// TIA Portal V16 export
// export: Created 2024-12-03T15:41:41.5093467Z, ExportSetting WithDefaults, DisplayName Totally Integrated Automation Portal, DisplayVersion V16 Update 6, DisplayName TIA Portal Version Control Interface, DisplayVersion V16 Update 2, DisplayName TIA Portal Openness, DisplayVersion V16 Update 6, DisplayName TIA Portal Teamcenter Gateway, DisplayVersion V16, DisplayName SINAMICS Startdrive Advanced, DisplayVersion V16 Update 5, DisplayName SINAMICS Startdrive G130, G150, S120, S150, SINAMICS MV, S210, DisplayVersion V16 Update 5, DisplayName SINAMICS Startdrive G110M, G120, G120C, G120D, G120P, G115D, DisplayVersion V16 Update 5, DisplayName STEP 7 Professional, DisplayVersion V16 Update 6, DisplayName STEP 7 Safety, DisplayVersion V16, DisplayName WinCC Advanced / Unified PC, DisplayVersion V16 Update 6
FUNCTION_BLOCK "ConveyLinxController_FullPLC"   // FB28, SCL
{ S7_Optimized_Access := 'FALSE' }
VERSION : 0.1
// stored: AutoNumber true, IsIECCheckEnabled false, SetENOAutomatically false, UDAEnableTagReadback false
   VAR_INPUT
      I_MotorData : "CLXAiPLC_IN_UDT";   // The 64 byte input word of the IO module
      I_RunOverride : Bool;
      I_OVerrideDirection : Bool;
      I_ControlLeftMotorConveyLInx : Bool;   // 1 = control left motor both motos can be controlled with one module
      I_ControlRightMotorConveyLinx : Bool;   // 1 = control right motor both motors can be controlled with one fb
   END_VAR
   VAR_IN_OUT
      IO_MotorStatus : "ConveyLinx_FullPLC_Single";
      IO_MotorOutput : "CLXAiPLC_OUT_UDT";   // All the motor commands
   END_VAR
   VAR DB_SPECIFIC
      S_NotConnected { S7_SetPoint := 'True'} : TON_TIME;
   END_VAR
   VAR
      cycleRun { S7_SetPoint := 'True'} : "CycleRun";
   END_VAR
   VAR DB_SPECIFIC
      AlarmInfo { S7_SetPoint := 'True'} : "AlarmInfo_UDT";
   END_VAR
   VAR
      Overheat { S7_SetPoint := 'True'} : Program_Alarm;
      ShortCircuit { S7_SetPoint := 'True'} : Program_Alarm;
      MDRNotConnected { S7_SetPoint := 'True'} : Program_Alarm;
      Overload { S7_SetPoint := 'True'} : Program_Alarm;
      Stalled { S7_SetPoint := 'True'} : Program_Alarm;
      MDRBadHall { S7_SetPoint := 'True'} : Program_Alarm;
      OverVoltage { S7_SetPoint := 'True'} : Program_Alarm;
      LowVoltage { S7_SetPoint := 'True'} : Program_Alarm;
      NotConnected { S7_SetPoint := 'True'} : Program_Alarm;
      ConnectionNotOK { S7_SetPoint := 'True'} : Program_Alarm;
      AnyErrorActive { S7_SetPoint := 'True'} : Program_Alarm;
      JamError { S7_SetPoint := 'True'} : Program_Alarm;
      SensorLowGain { S7_SetPoint := 'True'} : Program_Alarm;
   END_VAR
   VAR_TEMP
      T_AppState : "ApplicationState_UDT";
      T_ZoneInfo : "ZoneInfo";
   END_VAR
BEGIN
   #T_ZoneInfo := "ApplicationState_DB".ZoneNames[#IO_MotorStatus.Zone];
   #T_AppState := "ApplicationState_DB".Appstate[#T_ZoneInfo.AppStateIndex];
   #cycleRun(I_End:=13);

   REGION Commands

       #IO_MotorStatus.Status.ManualCommandsDisabled := 0;

       //Turn commands of if manual mode is deactivated
       IF NOT #T_AppState.States.ManualModeActivated.State THEN
           #IO_MotorStatus.Cmd.RunManual := 0;
           #IO_MotorStatus.Cmd.DirectionManual := 0;
           #IO_MotorStatus.Status.ManualCommandsDisabled := 1;
       END_IF;

       //Turn all commands of on error or interlock
       IF #IO_MotorStatus.Alarms.Status_1 > 0 OR #IO_MotorStatus.Status.Interlocked THEN
           #IO_MotorStatus.Cmd.RunAuto := 0;
           #IO_MotorStatus.Cmd.RunManual := 0;
           #IO_MotorStatus.Status.ManualCommandsDisabled := 1;
       END_IF;

       //Reset commands left
       IF #I_ControlLeftMotorConveyLInx THEN
           #IO_MotorOutput.LeftMDRControl.MDR_Direction := 0;
           #IO_MotorOutput.LeftMDRControl.Run_MDR := 0;
           #IO_MotorOutput.LeftMDRSpeed := 0;
           #IO_MotorOutput.ServoControlCommandLeft.RunToSetpoint := 0;
       END_IF;

       //Reset commands right
       IF #I_ControlRightMotorConveyLinx THEN
           #IO_MotorOutput.RightMDRControl.MDR_Direction := 0;
           #IO_MotorOutput.RightMDRControl.Run_MDR := 0;
           #IO_MotorOutput.RightMDRSpeed := 0;
           #IO_MotorOutput.ServoControlCommandRight.RunToSetpoint := 0;
       END_IF;

       //Auto mode left
       IF #T_AppState.States.AutoModeActivated.State
           AND #I_ControlLeftMotorConveyLInx THEN
           #IO_MotorOutput.LeftMDRControl.Run_MDR := #IO_MotorStatus.Cmd.RunAuto;
           #IO_MotorOutput.LeftMDRControl.MDR_Direction := #IO_MotorStatus.Cmd.DirectionAuto;
           #IO_MotorOutput.LeftMDRAccel := #IO_MotorStatus.Cmd.Accel;
           #IO_MotorOutput.LeftMDRDeccel := #IO_MotorStatus.Cmd.Deaccel;
           #IO_MotorOutput.LeftMDRSpeed := #IO_MotorStatus.Cmd.SpeedAuto;
           #IO_MotorOutput.LeftMDRBrakeMode := #IO_MotorStatus.Cmd.BrakeMode;
           #IO_MotorOutput.ServoControlCommandLeft.RunToSetpoint := #IO_MotorStatus.Cmd.ServoRunToSetpoint;
           #IO_MotorOutput.ServoControlCommandLeft.ResetPulseCount := #IO_MotorStatus.Cmd.ServoResetPulseCount;
           #IO_MotorOutput.LeftMDR_ServoMode := #IO_MotorStatus.Cmd.MDR_ServoMode;
           #IO_MotorOutput.ServoControlDistanceLeft := #IO_MotorStatus.Cmd.ServoControlDistance;
       END_IF;

       //Auto mode right
       IF #T_AppState.States.AutoModeActivated.State
           AND #I_ControlRightMotorConveyLinx THEN
           #IO_MotorOutput.RightMDRControl.Run_MDR := #IO_MotorStatus.Cmd.RunAuto;
           #IO_MotorOutput.RightMDRControl.MDR_Direction := #IO_MotorStatus.Cmd.DirectionAuto;
           #IO_MotorOutput.RightMDRAccel := #IO_MotorStatus.Cmd.Accel;
           #IO_MotorOutput.RightMDRDeccel := #IO_MotorStatus.Cmd.Deaccel;
           #IO_MotorOutput.RightMDRSpeed := #IO_MotorStatus.Cmd.SpeedAuto;
           #IO_MotorOutput.RightMDRBrakeMode := #IO_MotorStatus.Cmd.BrakeMode;
           #IO_MotorOutput.ServoControlCommandRight.RunToSetpoint := #IO_MotorStatus.Cmd.ServoRunToSetpoint;
           #IO_MotorOutput.ServoControlCommandRight.ResetPulseCount := #IO_MotorStatus.Cmd.ServoResetPulseCount;
           #IO_MotorOutput.RightMDR_ServoMode := #IO_MotorStatus.Cmd.MDR_ServoMode;
           #IO_MotorOutput.ServoControlDistanceRight := #IO_MotorStatus.Cmd.ServoControlDistance;
       END_IF;

       //Manual mode left
       IF #T_AppState.States.ManualModeActivated.State
           AND #I_ControlLeftMotorConveyLInx THEN
           IF NOT #IO_MotorStatus.Settings.AllowManualDirection THEN
               #IO_MotorOutput.LeftMDRControl.MDR_Direction := #IO_MotorStatus.Settings.DefaultDirection;
           ELSE
               #IO_MotorOutput.LeftMDRControl.MDR_Direction := #IO_MotorStatus.Cmd.DirectionManual;
           END_IF;
           #IO_MotorOutput.LeftMDRControl.Run_MDR := #IO_MotorStatus.Cmd.RunManual;
           #IO_MotorOutput.LeftMDRSpeed := #IO_MotorStatus.Cmd.SpeedManual;
       END_IF;

       //Manual mode right
       IF #T_AppState.States.ManualModeActivated.State
           AND #I_ControlRightMotorConveyLinx THEN

           IF NOT #IO_MotorStatus.Settings.AllowManualDirection THEN
               #IO_MotorOutput.RightMDRControl.MDR_Direction := #IO_MotorStatus.Settings.DefaultDirection;
           ELSE
               #IO_MotorOutput.RightMDRControl.MDR_Direction := #IO_MotorStatus.Cmd.DirectionManual;
           END_IF;

           #IO_MotorOutput.RightMDRControl.Run_MDR := #IO_MotorStatus.Cmd.RunManual;
           #IO_MotorOutput.RightMDRSpeed := #IO_MotorStatus.Cmd.SpeedManual;
       END_IF;

       REGION OVVERRIDE RUN
           IF #I_RunOverride THEN

               IF #I_ControlLeftMotorConveyLInx THEN
                   #IO_MotorOutput.LeftMDRControl.Run_MDR := true;
                   #IO_MotorOutput.LeftMDRControl.MDR_Direction := #I_OVerrideDirection;
                   #IO_MotorOutput.LeftMDRSpeed := 20;
               END_IF;

               IF #I_ControlRightMotorConveyLinx THEN
                   #IO_MotorOutput.RightMDRControl.Run_MDR := true;
                   #IO_MotorOutput.RightMDRControl.MDR_Direction := #I_OVerrideDirection;
                   #IO_MotorOutput.RightMDRSpeed := 20;
               END_IF;

           END_IF;

       END_REGION

   END_REGION

   REGION Interlock motor STATUS

       #IO_MotorStatus.Status.Interlocked := #IO_MotorStatus.Cmd.Interlock
       OR NOT #T_AppState.States.EmergencyOk.State;
       #IO_MotorStatus.Status.Status.%X0 := #IO_MotorStatus.Status.Interlocked;

   END_REGION

   REGION Create status

       //Left
       IF #I_ControlLeftMotorConveyLInx THEN
           #IO_MotorStatus.Status.ActualSpeed := #I_MotorData.LeftMDRRealSpeed;
           #IO_MotorStatus.Status.Current := #I_MotorData.LeftCurrent;
           #IO_MotorStatus.Status.Frequency := #I_MotorData.LeftFreq;
           #IO_MotorStatus.Status.ManualModeActive := #IO_MotorStatus.Cmd.RunManual;
           #IO_MotorStatus.Status.Position := #I_MotorData.DistanceLeft;
           #IO_MotorStatus.Status.Running := NOT #IO_MotorStatus.Alarms.AnyErrorActive.Active AND #IO_MotorOutput.LeftMDRControl.Run_MDR;
           #IO_MotorStatus.Status.ServoStatus.LastServoCommandExecuted := #I_MotorData.ServoStatusLeft.LastServoCommandExecuted;
           #IO_MotorStatus.Status.ServoStatus.ResetPulseCount_Echo := #I_MotorData.ServoStatusLeft.ResetPulseCount_Echo;
           #IO_MotorStatus.Status.ServoStatus.RunCommand_Echo := #I_MotorData.ServoStatusLeft.RunCommand_Echo;
           #IO_MotorStatus.Status.TemperatureModule := #I_MotorData.ModuleTemp;
           #IO_MotorStatus.Status.TeperatureMDR := #I_MotorData.LeftCalcTemp;
       END_IF;

       //right
       IF #I_ControlRightMotorConveyLinx THEN
           #IO_MotorStatus.Status.ActualSpeed := #I_MotorData.RightMDRRealSpeed;
           #IO_MotorStatus.Status.Current := #I_MotorData.RightCurrent;
           #IO_MotorStatus.Status.Frequency := #I_MotorData.RightFreq;
           #IO_MotorStatus.Status.ManualModeActive := #IO_MotorStatus.Cmd.RunManual;
           #IO_MotorStatus.Status.Position := #I_MotorData.DistanceRight;
           #IO_MotorStatus.Status.Running := NOT #IO_MotorStatus.Alarms.AnyErrorActive.Active AND #IO_MotorOutput.RightMDRControl.Run_MDR;
           #IO_MotorStatus.Status.ServoStatus.LastServoCommandExecuted := #I_MotorData.ServoStatusRight.LastServoCommandExecuted;
           #IO_MotorStatus.Status.ServoStatus.ResetPulseCount_Echo := #I_MotorData.ServoStatusRight.ResetPulseCount_Echo;
           #IO_MotorStatus.Status.ServoStatus.RunCommand_Echo := #I_MotorData.ServoStatusRight.RunCommand_Echo;
           #IO_MotorStatus.Status.TemperatureModule := #I_MotorData.ModuleTemp;
           #IO_MotorStatus.Status.TeperatureMDR := #I_MotorData.RightCalcTemp;
       END_IF;

       REGION Min max voltage

           #IO_MotorStatus.Status.Voltage := #I_MotorData.Voltage;
           IF #I_MotorData.Voltage < #IO_MotorStatus.Status.MinVoltage THEN
               #IO_MotorStatus.Status.MinVoltage := #I_MotorData.Voltage;
           END_IF;

           IF #I_MotorData.Voltage > #IO_MotorStatus.Status.MaxVoltage THEN
               #IO_MotorStatus.Status.MaxVoltage := #I_MotorData.Voltage;
           END_IF;

       END_REGION

       #IO_MotorStatus.Status.ManualModeActive := #T_AppState.States.ManualModeActivated.State;

       #IO_MotorStatus.Status.Status.%X1 := #IO_MotorStatus.Status.Running;
       #IO_MotorStatus.Status.Status.%X2 := #IO_MotorStatus.Status.ManualModeActive;

   END_REGION

   REGION Check alarm active

       IF #I_ControlLeftMotorConveyLInx THEN

           IF #I_MotorData.LeftMDRDiagnostic.LowVoltage THEN
               #IO_MotorStatus.Alarms.LowVoltage.Active := True;
           END_IF;

           IF #I_MotorData.LeftMDRDiagnostic.MDRBadHall THEN
               #IO_MotorStatus.Alarms.MDRBadHall.Active := True;
           END_IF;

           IF #I_MotorData.LeftMDRDiagnostic.MDRNotConnected THEN
               #IO_MotorStatus.Alarms.MDRNotConnected.Active := True;
           END_IF;

           IF #I_MotorData.LeftMDRDiagnostic.Overheat THEN
               #IO_MotorStatus.Alarms.Overheat.Active := True;
           END_IF;

           IF #I_MotorData.LeftMDRDiagnostic.Overload THEN
               #IO_MotorStatus.Alarms.Overload.Active := True;
           END_IF;

           IF #I_MotorData.LeftMDRDiagnostic.OverVoltage THEN
               #IO_MotorStatus.Alarms.OverVoltage.Active := True;
           END_IF;

           IF #I_MotorData.LeftMDRDiagnostic.ShortCircuit THEN
               #IO_MotorStatus.Alarms.ShortCircuit.Active := True;
           END_IF;

           IF #I_MotorData.LeftMDRDiagnostic.Stalled THEN
               #IO_MotorStatus.Alarms.Stalled.Active := True;
           END_IF;

       END_IF;

       IF #I_ControlRightMotorConveyLinx THEN

           IF #I_MotorData.RightMDRDiagnostic.LowVoltage THEN
               #IO_MotorStatus.Alarms.LowVoltage.Active := True;
           END_IF;

           IF #I_MotorData.RightMDRDiagnostic.MDRBadHall THEN
               #IO_MotorStatus.Alarms.MDRBadHall.Active := True;
           END_IF;

           IF #I_MotorData.RightMDRDiagnostic.MDRNotConnected THEN
               #IO_MotorStatus.Alarms.MDRNotConnected.Active := True;
           END_IF;

           IF #I_MotorData.RightMDRDiagnostic.Overheat THEN
               #IO_MotorStatus.Alarms.Overheat.Active := True;
           END_IF;

           IF #I_MotorData.RightMDRDiagnostic.Overload THEN
               #IO_MotorStatus.Alarms.Overload.Active := True;
           END_IF;

           IF #I_MotorData.RightMDRDiagnostic.OverVoltage THEN
               #IO_MotorStatus.Alarms.OverVoltage.Active := True;
           END_IF;

           IF #I_MotorData.RightMDRDiagnostic.ShortCircuit THEN
               #IO_MotorStatus.Alarms.ShortCircuit.Active := True;
           END_IF;

           IF #I_MotorData.RightMDRDiagnostic.Stalled THEN
               #IO_MotorStatus.Alarms.Stalled.Active := True;
           END_IF;

       END_IF;

       #IO_MotorStatus.Alarms.MDRBadHall.Active := FALSE;

       #IO_MotorStatus.Heartbeat := #I_MotorData.AllSensors.Heartbeat;
       #S_NotConnected(IN := NOT #IO_MotorStatus.Heartbeat,
                       PT := t#5s);

       IF #S_NotConnected.Q THEN
           #IO_MotorStatus.Alarms.NotConnected.Active := true;
       END_IF;

       REGION alarm info
           IF NOT #AlarmInfo.init OR "HMI_DB".ReloadSettings.signal THEN
               #IO_MotorStatus.Info.Name := "buildObjectName"(I_Symbolname := GetSymbolName(variable := #IO_MotorStatus, size := 100));
               #AlarmInfo.info := "buildAlarmInfo"(I_ZoneIndex := #IO_MotorStatus.Zone, I_ZoneName := #T_ZoneInfo.ZoneName, I_ObjectName := #IO_MotorStatus.Info.Name);
               #AlarmInfo.init := TRUE;
           END_IF;
       END_REGION

       REGION PROGRAM ALARMS

           IF #cycleRun.O_Cycle = 1 AND "RunTime_DB".CycleRun = #T_ZoneInfo.AppStateIndex THEN
               #Overheat(SIG := #IO_MotorStatus.Alarms.Overheat.Active,
                         SD_1 := #T_ZoneInfo.ZoneName,
                         SD_2 := #IO_MotorStatus.Info.Name,
                         SD_3 := #AlarmInfo.info);
           END_IF;

           IF #cycleRun.O_Cycle = 2 AND "RunTime_DB".CycleRun = #T_ZoneInfo.AppStateIndex THEN
               #ShortCircuit(SIG := #IO_MotorStatus.Alarms.ShortCircuit.Active,
                             SD_1 := #T_ZoneInfo.ZoneName,
                             SD_2 := #IO_MotorStatus.Info.Name,
                             SD_3 := #AlarmInfo.info);
           END_IF;

           IF #cycleRun.O_Cycle = 3 AND "RunTime_DB".CycleRun = #T_ZoneInfo.AppStateIndex THEN
               #MDRNotConnected(SIG := #IO_MotorStatus.Alarms.MDRNotConnected.Active,
                                SD_1 := #T_ZoneInfo.ZoneName,
                                SD_2 := #IO_MotorStatus.Info.Name,
                                SD_3 := #AlarmInfo.info);
           END_IF;

           IF #cycleRun.O_Cycle = 4 AND "RunTime_DB".CycleRun = #T_ZoneInfo.AppStateIndex THEN
               #Overload(SIG := #IO_MotorStatus.Alarms.Overload.Active,
                         SD_1 := #T_ZoneInfo.ZoneName,
                         SD_2 := #IO_MotorStatus.Info.Name,
                         SD_3 := #AlarmInfo.info);
           END_IF;

           IF #cycleRun.O_Cycle = 5 AND "RunTime_DB".CycleRun = #T_ZoneInfo.AppStateIndex THEN
               #Stalled(SIG := #IO_MotorStatus.Alarms.Stalled.Active,
                        SD_1 := #T_ZoneInfo.ZoneName,
                        SD_2 := #IO_MotorStatus.Info.Name,
                        SD_3 := #AlarmInfo.info);
           END_IF;

           IF #cycleRun.O_Cycle = 6 AND "RunTime_DB".CycleRun = #T_ZoneInfo.AppStateIndex THEN
               #MDRBadHall(SIG := #IO_MotorStatus.Alarms.MDRBadHall.Active,
                           SD_1 := #T_ZoneInfo.ZoneName,
                           SD_2 := #IO_MotorStatus.Info.Name,
                           SD_3 := #AlarmInfo.info);
           END_IF;

           IF #cycleRun.O_Cycle = 7 AND "RunTime_DB".CycleRun = #T_ZoneInfo.AppStateIndex THEN
               #OverVoltage(SIG := #IO_MotorStatus.Alarms.OverVoltage.Active,
                            SD_1 := #T_ZoneInfo.ZoneName,
                            SD_2 := #IO_MotorStatus.Info.Name,
                            SD_3 := #AlarmInfo.info);
           END_IF;

           IF #cycleRun.O_Cycle = 8 AND "RunTime_DB".CycleRun = #T_ZoneInfo.AppStateIndex THEN
               #LowVoltage(SIG := #IO_MotorStatus.Alarms.LowVoltage.Active,
                           SD_1 := #T_ZoneInfo.ZoneName,
                           SD_2 := #IO_MotorStatus.Info.Name,
                           SD_3 := #AlarmInfo.info);
           END_IF;

           IF #cycleRun.O_Cycle = 9 AND "RunTime_DB".CycleRun = #T_ZoneInfo.AppStateIndex THEN
               #NotConnected(SIG := #IO_MotorStatus.Alarms.NotConnected.Active,
                             SD_1 := #T_ZoneInfo.ZoneName,
                             SD_2 := #IO_MotorStatus.Info.Name,
                             SD_3 := #AlarmInfo.info);
           END_IF;

           IF #cycleRun.O_Cycle = 10 AND "RunTime_DB".CycleRun = #T_ZoneInfo.AppStateIndex THEN
               #ConnectionNotOK(SIG := #IO_MotorStatus.Alarms.ConnectionNotOK.Active,
                                SD_1 := #T_ZoneInfo.ZoneName,
                                SD_2 := #IO_MotorStatus.Info.Name,
                                SD_3 := #AlarmInfo.info);
           END_IF;


           IF #cycleRun.O_Cycle = 11 AND "RunTime_DB".CycleRun = #T_ZoneInfo.AppStateIndex THEN
               #AnyErrorActive(SIG := #IO_MotorStatus.Alarms.AnyErrorActive.Active,
                               SD_1 := #T_ZoneInfo.ZoneName,
                               SD_2 := #IO_MotorStatus.Info.Name,
                               SD_3 := #AlarmInfo.info);
           END_IF;

           IF #cycleRun.O_Cycle = 12 AND "RunTime_DB".CycleRun = #T_ZoneInfo.AppStateIndex THEN
               #JamError(SIG := #IO_MotorStatus.Alarms.JamError.Active,
                         SD_1 := #T_ZoneInfo.ZoneName,
                         SD_2 := #IO_MotorStatus.Info.Name,
                         SD_3 := #AlarmInfo.info);
           END_IF;

           IF #cycleRun.O_Cycle = 13 AND "RunTime_DB".CycleRun = #T_ZoneInfo.AppStateIndex THEN
               #SensorLowGain(SIG := #IO_MotorStatus.Alarms.SensorLowGain.Active,
                              SD_1 := #T_ZoneInfo.ZoneName,
                              SD_2 := #IO_MotorStatus.Info.Name,
                              SD_3 := #AlarmInfo.info);
           END_IF;
       END_REGION

   END_REGION

   REGION Alarm status

       #IO_MotorStatus.Alarms.Status_1.%X0 := #IO_MotorStatus.Alarms.Overheat.Active;
       //#MotorStatus.Alarms.Status_1.%X1 := #MotorStatus.Alarms.Overheat.Active;
       #IO_MotorStatus.Alarms.Status_1.%X2 := #IO_MotorStatus.Alarms.ShortCircuit.Active;
       #IO_MotorStatus.Alarms.Status_1.%X3 := #IO_MotorStatus.Alarms.MDRNotConnected.Active;

       #IO_MotorStatus.Alarms.Status_1.%X4 := #IO_MotorStatus.Alarms.Overload.Active;
       #IO_MotorStatus.Alarms.Status_1.%X5 := #IO_MotorStatus.Alarms.Stalled.Active;
       #IO_MotorStatus.Alarms.Status_1.%X6 := #IO_MotorStatus.Alarms.MDRBadHall.Active;
       // #MotorStatus.Alarms.Status_1.%X7 := #MotorStatus.Alarms.Overheat.Active;

       #IO_MotorStatus.Alarms.Status_1.%X8 := #IO_MotorStatus.Alarms.OverVoltage.Active;
       #IO_MotorStatus.Alarms.Status_1.%X9 := #IO_MotorStatus.Alarms.LowVoltage.Active;
       #IO_MotorStatus.Alarms.Status_1.%X10 := #IO_MotorStatus.Alarms.NotConnected.Active;
       #IO_MotorStatus.Alarms.Status_1.%X11 := #IO_MotorStatus.Alarms.ConnectionNotOK.Active;

       #IO_MotorStatus.Alarms.Status_1.%X12 := #IO_MotorStatus.Alarms.AnyErrorActive.Active;
       #IO_MotorStatus.Alarms.Status_1.%X13 := #IO_MotorStatus.Alarms.JamError.Active;
       #IO_MotorStatus.Alarms.Status_1.%X14 := #IO_MotorStatus.Alarms.SensorLowGain.Active;
       //#MotorStatus.Alarms.Status_1.%X15 := #MotorStatus.Alarms.Overheat.Active;

       IF #IO_MotorStatus.Alarms.Status_1 > 0 THEN
           "ApplicationState_DB".Appstate[#T_ZoneInfo.AppStateIndex].Alarms.AlarmActiveInternalPLC := TRUE;
       END_IF;

   END_REGION

   REGION Reset alarms

       IF #IO_MotorStatus.Alarms.Status_1 > 0
           AND (#T_AppState.Hmi_Buttons.reset.state.State OR #IO_MotorStatus.Cmd.Reset OR "Simulation_DB".Simulation_On)
           OR #I_RunOverride THEN

           #IO_MotorStatus.Alarms.Overheat.Active := False;
           #IO_MotorStatus.Alarms.Overheat.Active := False;
           #IO_MotorStatus.Alarms.ShortCircuit.Active := False;
           #IO_MotorStatus.Alarms.MDRNotConnected.Active := False;

           #IO_MotorStatus.Alarms.Overload.Active := False;
           #IO_MotorStatus.Alarms.Stalled.Active := False;
           #IO_MotorStatus.Alarms.MDRBadHall.Active := False;
           #IO_MotorStatus.Alarms.Overheat.Active := False;
           #IO_MotorStatus.Alarms.OverVoltage.Active := False;
           #IO_MotorStatus.Alarms.LowVoltage.Active := False;
           #IO_MotorStatus.Alarms.NotConnected.Active := False;
           #IO_MotorStatus.Alarms.ConnectionNotOK.Active := False;

           #IO_MotorStatus.Alarms.AnyErrorActive.Active := False;
           #IO_MotorStatus.Alarms.JamError.Active := False;
           #IO_MotorStatus.Alarms.SensorLowGain.Active := False;
           #IO_MotorStatus.Alarms.Overheat.Active := False;

       END_IF;

   END_REGION

   REGION common status
       #IO_MotorStatus.Info.CommonStatus := 0;
       IF #IO_MotorStatus.Status.Running THEN
           #IO_MotorStatus.Info.CommonStatus := 1;
       END_IF;

       IF #IO_MotorStatus.Alarms.Status_1 > 1 THEN
           #IO_MotorStatus.Info.CommonStatus := 2;
       END_IF;
   END_REGION

   #IO_MotorStatus.Cmd.Reset := 0;
END_FUNCTION_BLOCK
